(* Logix 5000 project; controller R5_CSS vendor 1 type 14 code 74 rev 19.11; software revision 19.01; part 7 of 20 *)
(* tags used below, declared in another part *)
   AC102A : ANALYTICAL;   // QUENCH WATER CONDUCTIVITY CONTROL
   AC102A_BLEED_MAKEUP_STATUS : DINT;   // 0=stopped 1=bleed water 2=makeup water 3=wait
   AC102A_BLEED_START_TON : TIMER;
   AC102A_BLEED_STOP_TON : TIMER;
   AC102A_BLEED_WAIT : BOOL;
   AC102A_BLEED_WAIT_TON : TIMER;
   AC102A_MAKEUP_STOP_TON : TIMER;
   AlarmMaster : DINT;
   AlarmsAckAll : BOOL;
   AlarmsDisabled : BOOL;
   F1_LC370 : LEVEL_CONTROL;
   FC141 : PUMP_CONTROL;
   FC215 : FLOW_CONTROL;   // OVERHEAD CONDENSER CHILLED WATER FLOW CONTROL
   FC365 : FLOW_CONTROL;   // COALESCER PROCESS IMPURITY FLOW CONTROL
   FC365_Alm : ALARM_ANALOG;
   FC365_AUTO_ONS1 : BOOL;
   FC365_AUTO_ONS2 : BOOL;
   FC365_BLEED_ALARM_DISABLE : BOOL;
   FC365_BLEED_FLOW_MIN_SP : DINT;
   FC365_BLEED_WAIT_MIN_SP : DINT;
   FC365_FLOW_TOO_LONG_ALM : BOOL;
   FC365_FLOW_TOO_LONG_RESETPB : BOOL;
   FC365_FLOW_TOO_LONG_TMR : TIMER;
   FC365_HMI_BLEED_START_ENABLE : BOOL;
   FC365_HMI_BLEED_START_ENABLE_TON : TIMER;
   FC365_HMI_BLEED_START_PB : BOOL;
   FC365_HMI_BLEED_STOP_PB : BOOL;
   FC365_LC370_FLOW_AUTO_SP : REAL;
   FC365_MANUAL_ONS1 : BOOL;
   FC365_MAX_TIME_MIN : DINT;
   FC365_Started : BOOL;
   FC365_TOTAl_GAL : REAL;
   FC365_TOTAl_RESET : BOOL;
   FC365_TOTAl_RESET_PB : BOOL;
   FC365_TOTALIZE : Totalize;
   FC365_TOTALIZE_EN : BOOL;
   FC365_TOTALIZE_EN_ONS1 : BOOL;
   FC365_TOTALIZE_LastFeedTimeMin : REAL;
   FC365_TOTALIZE_Min : REAL;
   FC365_TOTALIZE_TON : TIMER;
   FC365_UNABLE_TO_BLEED : BOOL;
   FC370 : FLOW_CONTROL;   // COALESCER MAKE UP WATER FLOW CONTROL
   FC403 : FLOW_CONTROL;   // COALESCER FLOW CONTROLLER FEEDS TCV108
   FC406 : FLOW_CONTROL;   // HX COOLING WATER FLOW CONTROL
   FCV141_MaxOpenSecSP : REAL;
   FCV141_MaxOpenTmr : TIMER;
   FireFlowAlarmFromUTL : BOOL;
   HS141 : ValveControl_TwoWay;
   InputMax_IF8 : REAL;
   InputMin_IF8 : REAL;
   LC303A : LEVEL_CONTROL;   // AQUEOUS PHASE OF PRIMARY SETTLER
   LC303B : LEVEL_CONTROL;   // INTERFACE LEVEL OF PRIMARY CONDENSER
   LC365_AUTO_SP_START : REAL;
   LC365_BLEED_AUTO_START : BOOL;
   LC365_BLEED_AUTO_START_TON : TIMER;
   LC365_LT : REAL;
   LC370 : LEVEL_CONTROL;   // WATER MAKE UP FOR PRIMARY SETTLER
   LC370_AUTO_SP_START : REAL;
   LCV370_Start : BOOL;
   PID_FCV365 : PID;
   PID_FCV365_TON : TIMER;
   PID_LC370_Enable : BOOL;
   SignalLossHigh_IF8 : DINT;
   SignalLossLow_IF8 : DINT;
   TC313A : TEMP_CONTROL;   // PRIMARY COALESCER SEPARATOR TEMPERATURE CONTROL
   TMR_FAULT : DINT;
   UTL_Comms : DINT[3];
(* MainProgram, continued *)

ROUTINE FC215_OverheadCondChillWaterFlow   (* ladder *)
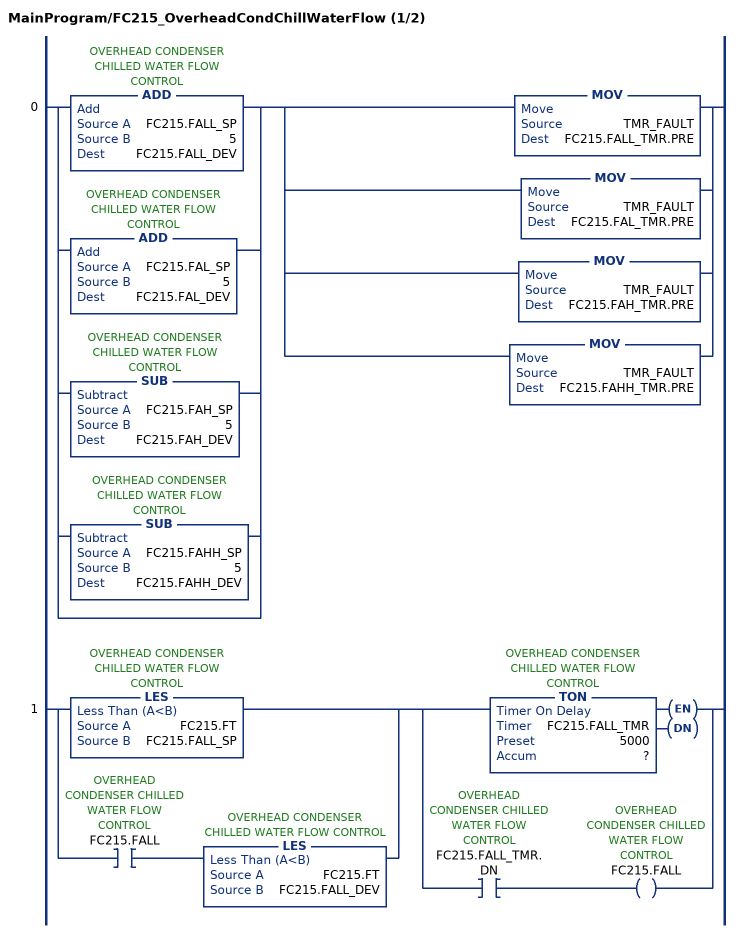
   0: [ADD(FC215.FALL_SP,5,FC215.FALL_DEV) ,ADD(FC215.FAL_SP,5,FC215.FAL_DEV) ,SUB(FC215.FAH_SP,5,FC215.FAH_DEV) ,SUB(FC215.FAHH_SP,5,FC215.FAHH_DEV) ,][MOV(TMR_FAULT,FC215.FALL_TMR.PRE) ,MOV(TMR_FAULT,FC215.FAL_TMR.PRE) ,MOV(TMR_FAULT,FC215.FAH_TMR.PRE) ,MOV(TMR_FAULT,FC215.FAHH_TMR.PRE) ];
   1: [LES(FC215.FT,FC215.FALL_SP) ,XIC(FC215.FALL) LES(FC215.FT,FC215.FALL_DEV) ][TON(FC215.FALL_TMR,?,?) ,XIC(FC215.FALL_TMR.DN) OTE(FC215.FALL) ];
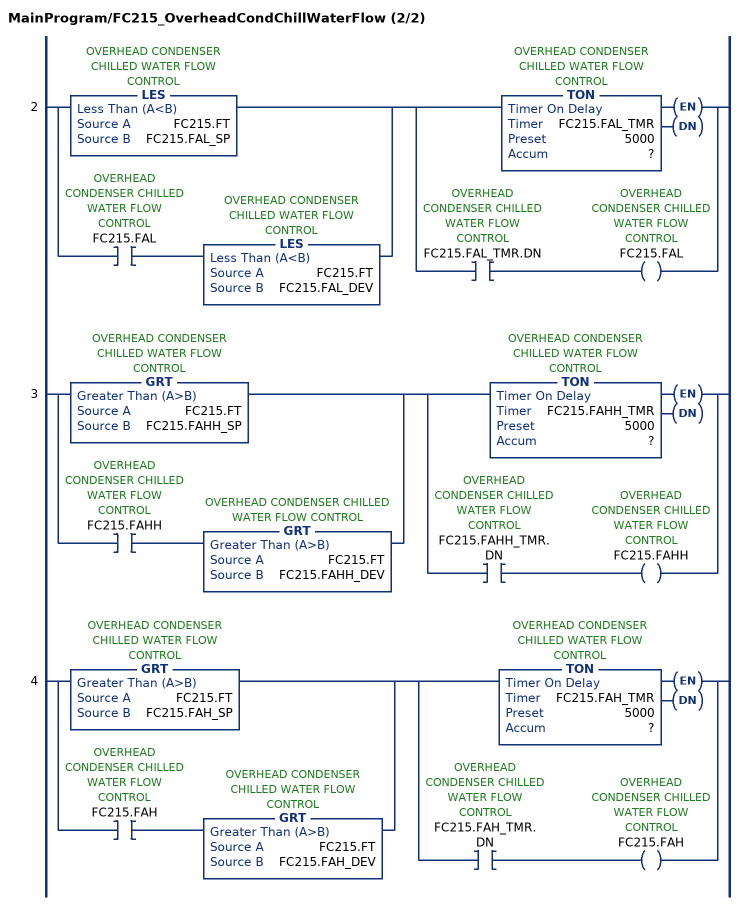
   2: [LES(FC215.FT,FC215.FAL_SP) ,XIC(FC215.FAL) LES(FC215.FT,FC215.FAL_DEV) ][TON(FC215.FAL_TMR,?,?) ,XIC(FC215.FAL_TMR.DN) OTE(FC215.FAL) ];
   3: [GRT(FC215.FT,FC215.FAHH_SP) ,XIC(FC215.FAHH) GRT(FC215.FT,FC215.FAHH_DEV) ][TON(FC215.FAHH_TMR,?,?) ,XIC(FC215.FAHH_TMR.DN) OTE(FC215.FAHH) ];
   4: [GRT(FC215.FT,FC215.FAH_SP) ,XIC(FC215.FAH) GRT(FC215.FT,FC215.FAH_DEV) ][TON(FC215.FAH_TMR,?,?) ,XIC(FC215.FAH_TMR.DN) OTE(FC215.FAH) ];
END_ROUTINE

ROUTINE FC370_WaterMakeupFlow   (* ladder *)
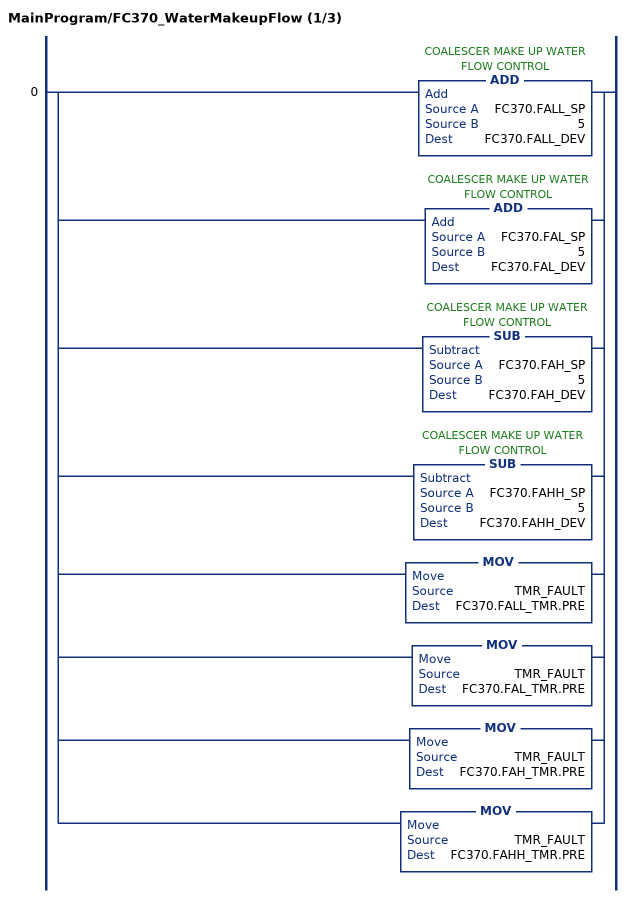
   0: [ADD(FC370.FALL_SP,5,FC370.FALL_DEV) ,ADD(FC370.FAL_SP,5,FC370.FAL_DEV) ,SUB(FC370.FAH_SP,5,FC370.FAH_DEV) ,SUB(FC370.FAHH_SP,5,FC370.FAHH_DEV) ,MOV(TMR_FAULT,FC370.FALL_TMR.PRE) ,MOV(TMR_FAULT,FC370.FAL_TMR.PRE) ,MOV(TMR_FAULT,FC370.FAH_TMR.PRE) ,MOV(TMR_FAULT,FC370.FAHH_TMR.PRE) ];
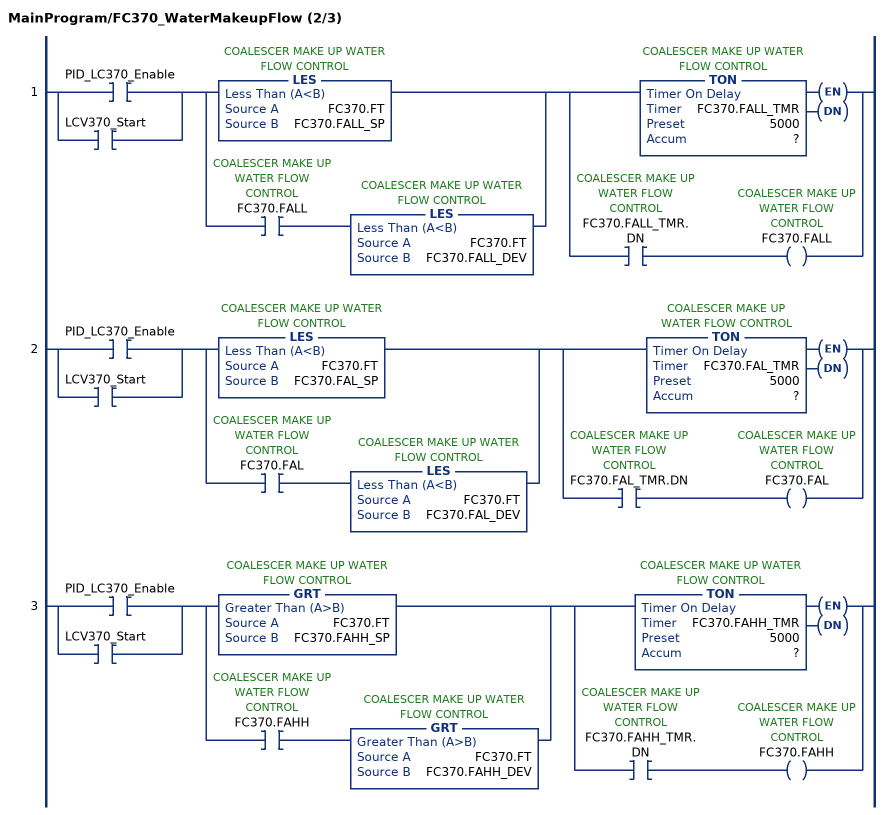
   1: [XIC(PID_LC370_Enable) ,XIC(LCV370_Start) ][LES(FC370.FT,FC370.FALL_SP) ,XIC(FC370.FALL) LES(FC370.FT,FC370.FALL_DEV) ][TON(FC370.FALL_TMR,?,?) ,XIC(FC370.FALL_TMR.DN) OTE(FC370.FALL) ];
   2: [XIC(PID_LC370_Enable) ,XIC(LCV370_Start) ][LES(FC370.FT,FC370.FAL_SP) ,XIC(FC370.FAL) LES(FC370.FT,FC370.FAL_DEV) ][TON(FC370.FAL_TMR,?,?) ,XIC(FC370.FAL_TMR.DN) OTE(FC370.FAL) ];
   3: [XIC(PID_LC370_Enable) ,XIC(LCV370_Start) ][GRT(FC370.FT,FC370.FAHH_SP) ,XIC(FC370.FAHH) GRT(FC370.FT,FC370.FAHH_DEV) ][TON(FC370.FAHH_TMR,?,?) ,XIC(FC370.FAHH_TMR.DN) OTE(FC370.FAHH) ];
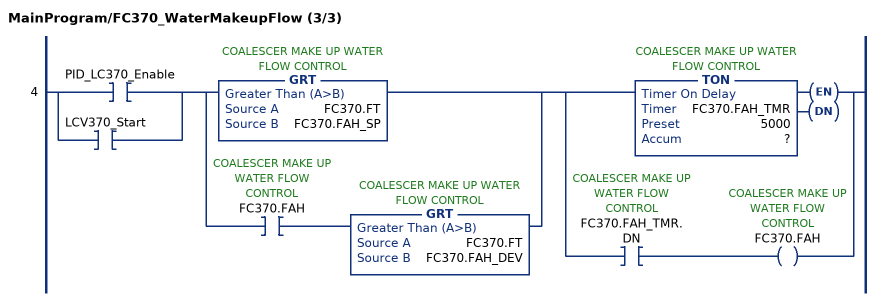
   4: [XIC(PID_LC370_Enable) ,XIC(LCV370_Start) ][GRT(FC370.FT,FC370.FAH_SP) ,XIC(FC370.FAH) GRT(FC370.FT,FC370.FAH_DEV) ][TON(FC370.FAH_TMR,?,?) ,XIC(FC370.FAH_TMR.DN) OTE(FC370.FAH) ];
END_ROUTINE

ROUTINE FC403_QuenchWaterTotalFlow   (* ladder *)
// COALESCER FLOW CONTROL
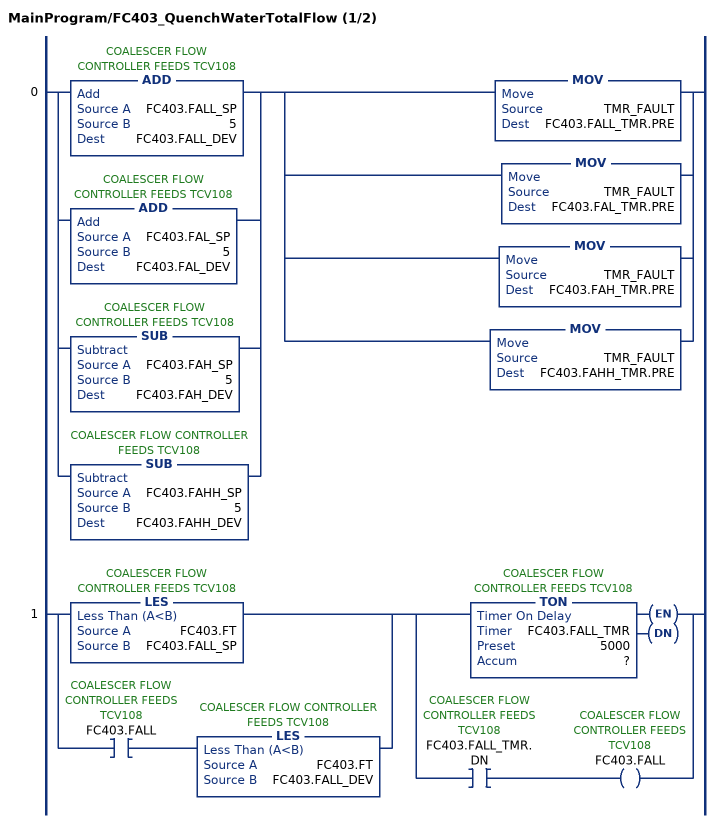
   0: [ADD(FC403.FALL_SP,5,FC403.FALL_DEV) ,ADD(FC403.FAL_SP,5,FC403.FAL_DEV) ,SUB(FC403.FAH_SP,5,FC403.FAH_DEV) ,SUB(FC403.FAHH_SP,5,FC403.FAHH_DEV) ][MOV(TMR_FAULT,FC403.FALL_TMR.PRE) ,MOV(TMR_FAULT,FC403.FAL_TMR.PRE) ,MOV(TMR_FAULT,FC403.FAH_TMR.PRE) ,MOV(TMR_FAULT,FC403.FAHH_TMR.PRE) ];
   1: [LES(FC403.FT,FC403.FALL_SP) ,XIC(FC403.FALL) LES(FC403.FT,FC403.FALL_DEV) ][TON(FC403.FALL_TMR,?,?) ,XIC(FC403.FALL_TMR.DN) OTE(FC403.FALL) ];
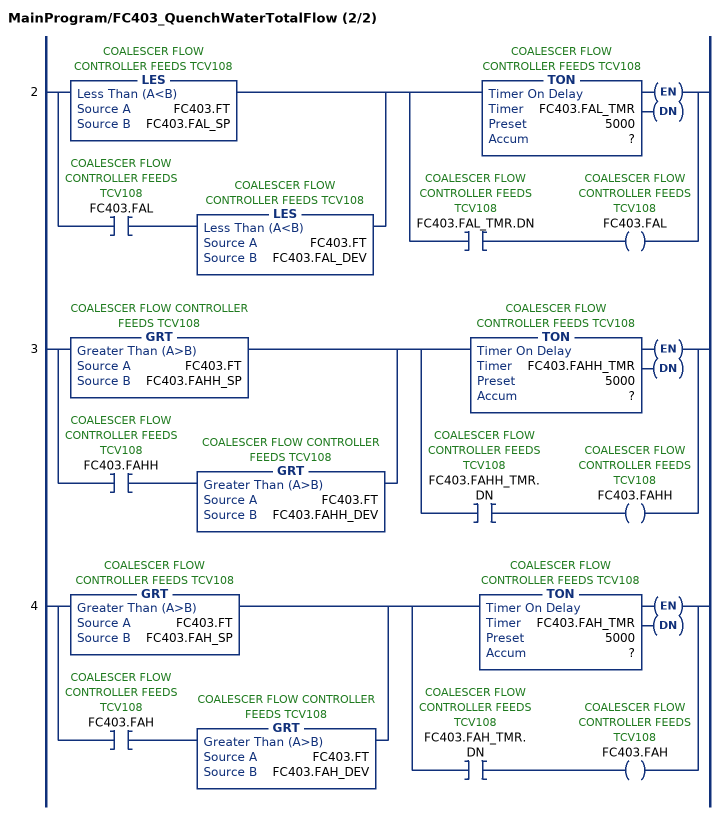
   2: [LES(FC403.FT,FC403.FAL_SP) ,XIC(FC403.FAL) LES(FC403.FT,FC403.FAL_DEV) ][TON(FC403.FAL_TMR,?,?) ,XIC(FC403.FAL_TMR.DN) OTE(FC403.FAL) ];
   3: [GRT(FC403.FT,FC403.FAHH_SP) ,XIC(FC403.FAHH) GRT(FC403.FT,FC403.FAHH_DEV) ][TON(FC403.FAHH_TMR,?,?) ,XIC(FC403.FAHH_TMR.DN) OTE(FC403.FAHH) ];
   4: [GRT(FC403.FT,FC403.FAH_SP) ,XIC(FC403.FAH) GRT(FC403.FT,FC403.FAH_DEV) ][TON(FC403.FAH_TMR,?,?) ,XIC(FC403.FAH_TMR.DN) OTE(FC403.FAH) ];
END_ROUTINE

ROUTINE FC406_CoolingWaterFlow   (* ladder *)
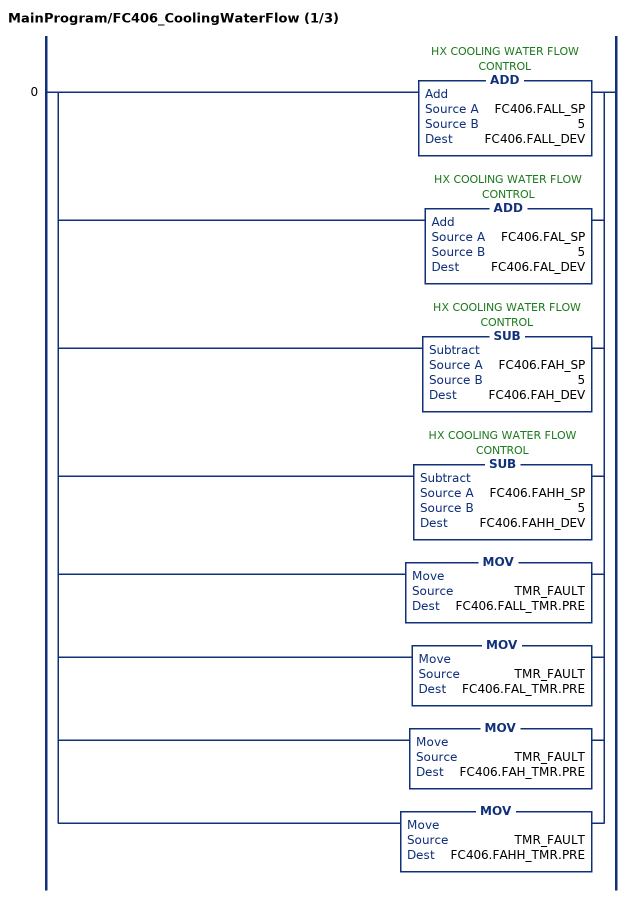
   0: [ADD(FC406.FALL_SP,5,FC406.FALL_DEV) ,ADD(FC406.FAL_SP,5,FC406.FAL_DEV) ,SUB(FC406.FAH_SP,5,FC406.FAH_DEV) ,SUB(FC406.FAHH_SP,5,FC406.FAHH_DEV) ,MOV(TMR_FAULT,FC406.FALL_TMR.PRE) ,MOV(TMR_FAULT,FC406.FAL_TMR.PRE) ,MOV(TMR_FAULT,FC406.FAH_TMR.PRE) ,MOV(TMR_FAULT,FC406.FAHH_TMR.PRE) ];
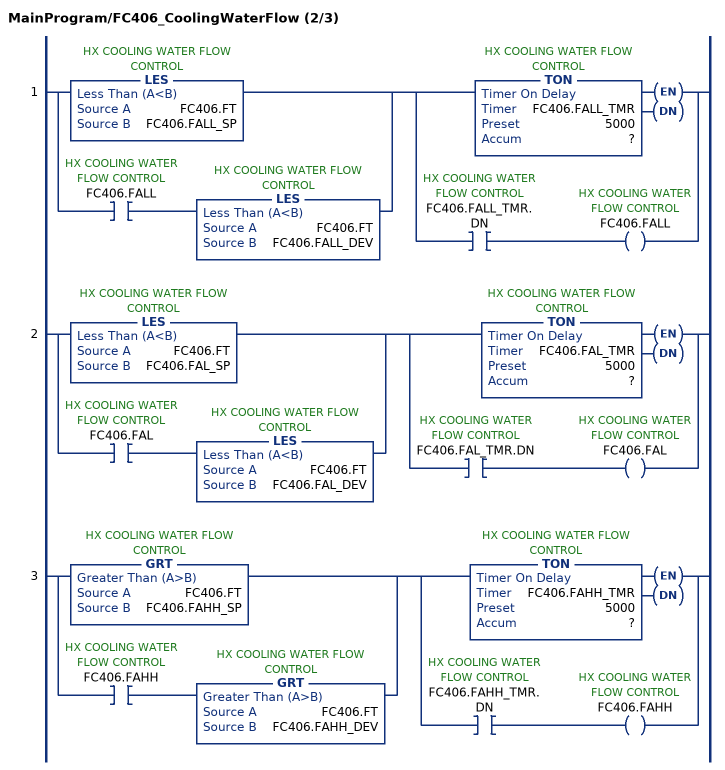
   1: [LES(FC406.FT,FC406.FALL_SP) ,XIC(FC406.FALL) LES(FC406.FT,FC406.FALL_DEV) ][TON(FC406.FALL_TMR,?,?) ,XIC(FC406.FALL_TMR.DN) OTE(FC406.FALL) ];
   2: [LES(FC406.FT,FC406.FAL_SP) ,XIC(FC406.FAL) LES(FC406.FT,FC406.FAL_DEV) ][TON(FC406.FAL_TMR,?,?) ,XIC(FC406.FAL_TMR.DN) OTE(FC406.FAL) ];
   3: [GRT(FC406.FT,FC406.FAHH_SP) ,XIC(FC406.FAHH) GRT(FC406.FT,FC406.FAHH_DEV) ][TON(FC406.FAHH_TMR,?,?) ,XIC(FC406.FAHH_TMR.DN) OTE(FC406.FAHH) ];
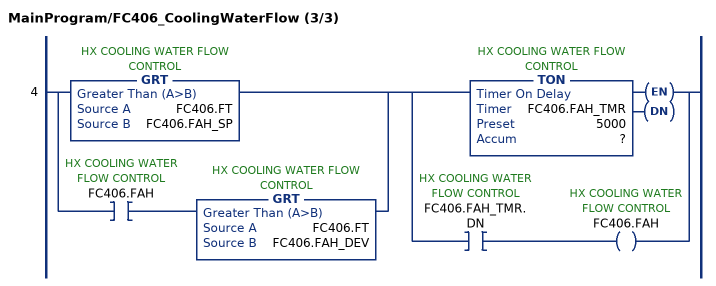
   4: [GRT(FC406.FT,FC406.FAH_SP) ,XIC(FC406.FAH) GRT(FC406.FT,FC406.FAH_DEV) ][TON(FC406.FAH_TMR,?,?) ,XIC(FC406.FAH_TMR.DN) OTE(FC406.FAH) ];
END_ROUTINE

ROUTINE FCV141_QuenchTowerEmegencyValve   (* ladder *)
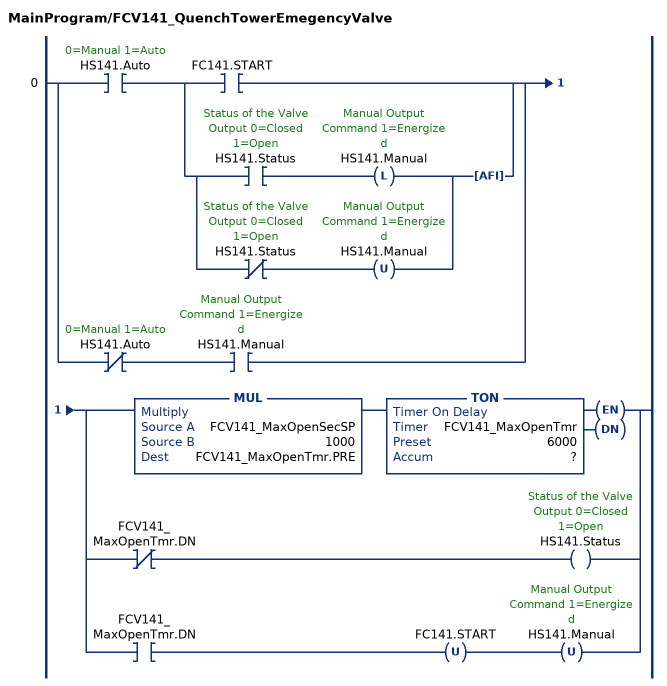
   0: [XIC(HS141.Auto) [XIC(FC141.START) ,[XIC(HS141.Status) OTL(HS141.Manual) ,XIO(HS141.Status) OTU(HS141.Manual) ] AFI() ] ,XIO(HS141.Auto) XIC(HS141.Manual) ][MUL(FCV141_MaxOpenSecSP,1000,FCV141_MaxOpenTmr.PRE) TON(FCV141_MaxOpenTmr,?,?) ,XIO(FCV141_MaxOpenTmr.DN) OTE(HS141.Status) ,XIC(FCV141_MaxOpenTmr.DN) OTU(FC141.START) OTU(HS141.Manual) ];
END_ROUTINE

ROUTINE FCV365_WaterBleedLevel_PID   (* ladder *)
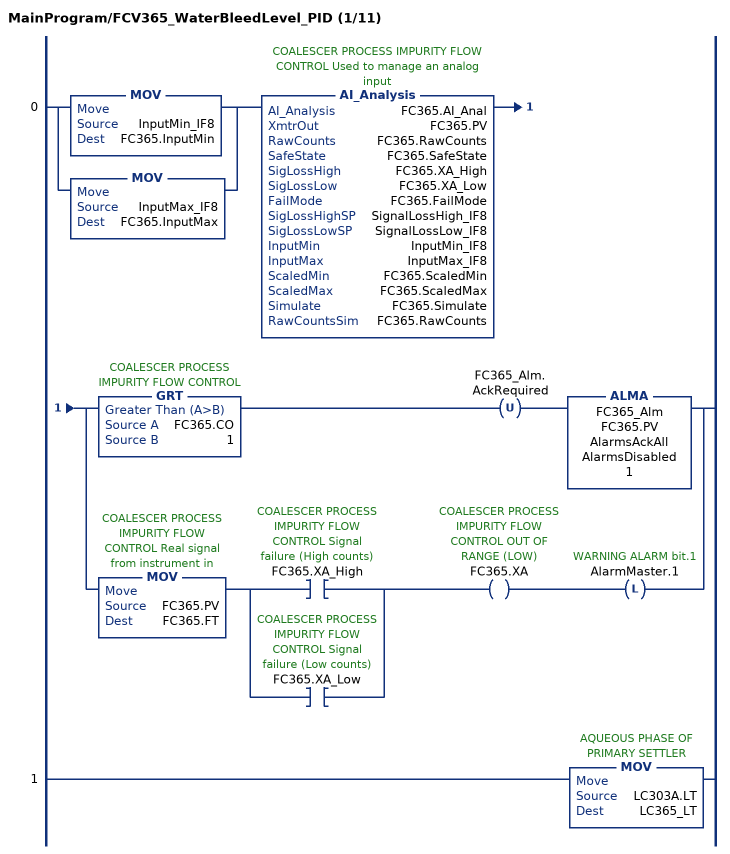
   0: [MOV(InputMin_IF8,FC365.InputMin) ,MOV(InputMax_IF8,FC365.InputMax) ]AI_Analysis(FC365.AI_Anal,FC365.PV,FC365.RawCounts,FC365.SafeState,FC365.XA_High,FC365.XA_Low,FC365.FailMode,SignalLossHigh_IF8,SignalLossLow_IF8,InputMin_IF8,InputMax_IF8,FC365.ScaledMin,FC365.ScaledMax,FC365.Simulate,FC365.RawCounts)[GRT(FC365.CO,1) OTU(FC365_Alm.AckRequired) ALMA(FC365_Alm,FC365.PV,AlarmsAckAll,AlarmsDisabled,1) ,MOV(FC365.PV,FC365.FT) [XIC(FC365.XA_High) ,XIC(FC365.XA_Low) ] OTE(FC365.XA) OTL(AlarmMaster.1) ];
   1: MOV(LC303A.LT,LC365_LT);
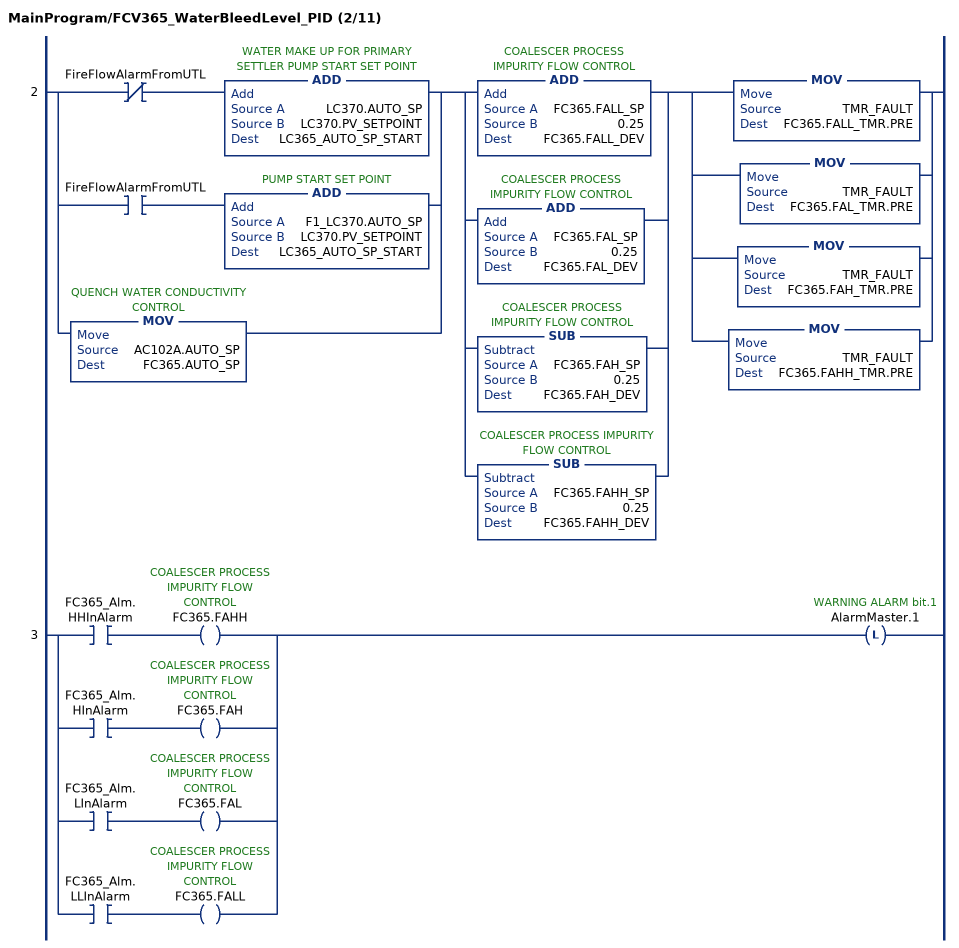
   2: [XIO(FireFlowAlarmFromUTL) ADD(LC370.AUTO_SP,LC370.PV_SETPOINT,LC365_AUTO_SP_START) ,XIC(FireFlowAlarmFromUTL) ADD(F1_LC370.AUTO_SP,LC370.PV_SETPOINT,LC365_AUTO_SP_START) ,MOV(AC102A.AUTO_SP,FC365.AUTO_SP) ][ADD(FC365.FALL_SP,0.25,FC365.FALL_DEV) ,ADD(FC365.FAL_SP,0.25,FC365.FAL_DEV) ,SUB(FC365.FAH_SP,0.25,FC365.FAH_DEV) ,SUB(FC365.FAHH_SP,0.25,FC365.FAHH_DEV) ][MOV(TMR_FAULT,FC365.FALL_TMR.PRE) ,MOV(TMR_FAULT,FC365.FAL_TMR.PRE) ,MOV(TMR_FAULT,FC365.FAH_TMR.PRE) ,MOV(TMR_FAULT,FC365.FAHH_TMR.PRE) ];
   3: [XIC(FC365_Alm.HHInAlarm) OTE(FC365.FAHH) ,XIC(FC365_Alm.HInAlarm) OTE(FC365.FAH) ,XIC(FC365_Alm.LInAlarm) OTE(FC365.FAL) ,XIC(FC365_Alm.LLInAlarm) OTE(FC365.FALL) ]OTL(AlarmMaster.1);
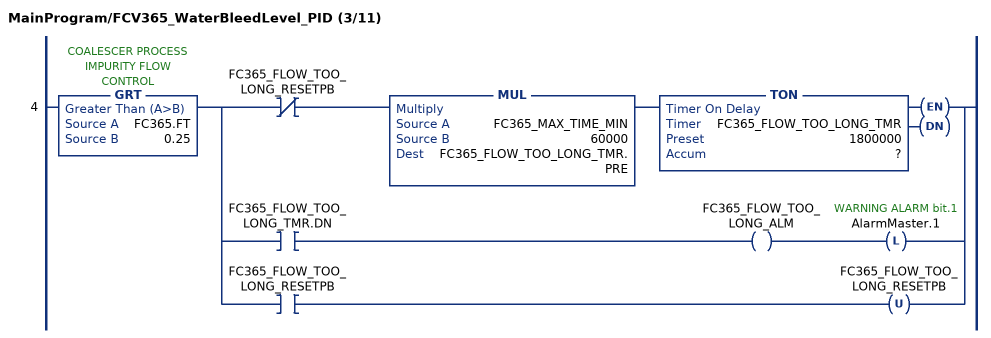
   4: GRT(FC365.FT,0.25)[XIO(FC365_FLOW_TOO_LONG_RESETPB) MUL(FC365_MAX_TIME_MIN,60000,FC365_FLOW_TOO_LONG_TMR.PRE) TON(FC365_FLOW_TOO_LONG_TMR,?,?) ,XIC(FC365_FLOW_TOO_LONG_TMR.DN) OTE(FC365_FLOW_TOO_LONG_ALM) OTL(AlarmMaster.1) ,XIC(FC365_FLOW_TOO_LONG_RESETPB) OTU(FC365_FLOW_TOO_LONG_RESETPB) ];
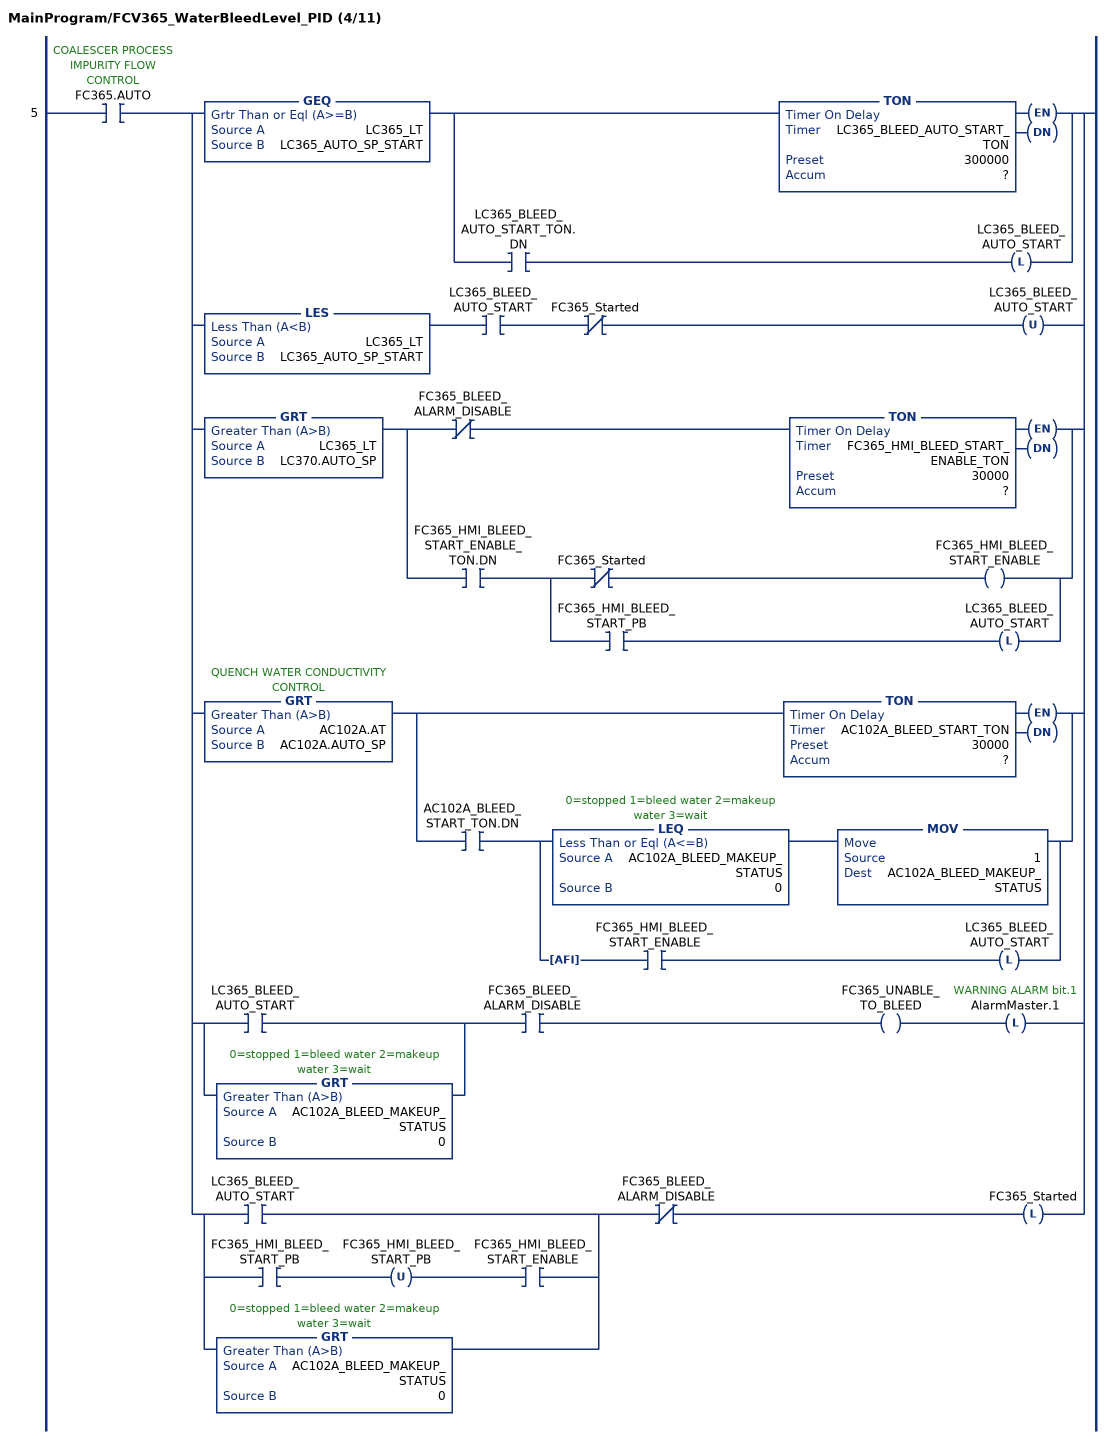
   5: XIC(FC365.AUTO)[GEQ(LC365_LT,LC365_AUTO_SP_START) [TON(LC365_BLEED_AUTO_START_TON,?,?) ,XIC(LC365_BLEED_AUTO_START_TON.DN) OTL(LC365_BLEED_AUTO_START) ] ,LES(LC365_LT,LC365_AUTO_SP_START) XIC(LC365_BLEED_AUTO_START) XIO(FC365_Started) OTU(LC365_BLEED_AUTO_START) ,GRT(LC365_LT,LC370.AUTO_SP) [XIO(FC365_BLEED_ALARM_DISABLE) TON(FC365_HMI_BLEED_START_ENABLE_TON,?,?) ,XIC(FC365_HMI_BLEED_START_ENABLE_TON.DN) [XIO(FC365_Started) OTE(FC365_HMI_BLEED_START_ENABLE) ,XIC(FC365_HMI_BLEED_START_PB) OTL(LC365_BLEED_AUTO_START) ] ] ,GRT(AC102A.AT,AC102A.AUTO_SP) [TON(AC102A_BLEED_START_TON,?,?) ,XIC(AC102A_BLEED_START_TON.DN) [LEQ(AC102A_BLEED_MAKEUP_STATUS,0) MOV(1,AC102A_BLEED_MAKEUP_STATUS) ,AFI() XIC(FC365_HMI_BLEED_START_ENABLE) OTL(LC365_BLEED_AUTO_START) ] ] ,[XIC(LC365_BLEED_AUTO_START) ,GRT(AC102A_BLEED_MAKEUP_STATUS,0) ] XIC(FC365_BLEED_ALARM_DISABLE) OTE(FC365_UNABLE_TO_BLEED) OTL(AlarmMaster.1) ,[XIC(LC365_BLEED_AUTO_START) ,XIC(FC365_HMI_BLEED_START_PB) OTU(FC365_HMI_BLEED_START_PB) XIC(FC365_HMI_BLEED_START_ENABLE) ,GRT(AC102A_BLEED_MAKEUP_STATUS,0) ] XIO(FC365_BLEED_ALARM_DISABLE) OTL(FC365_Started) ];
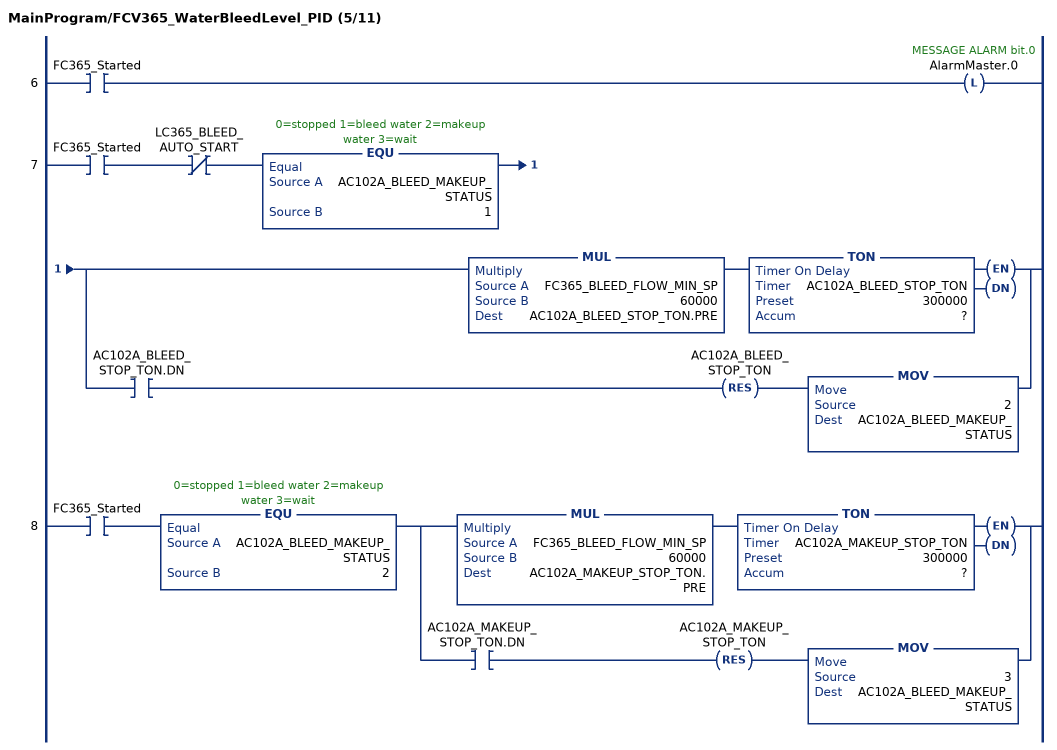
   6: XIC(FC365_Started)OTL(AlarmMaster.0);
   7: XIC(FC365_Started)XIO(LC365_BLEED_AUTO_START)EQU(AC102A_BLEED_MAKEUP_STATUS,1)[MUL(FC365_BLEED_FLOW_MIN_SP,60000,AC102A_BLEED_STOP_TON.PRE) TON(AC102A_BLEED_STOP_TON,?,?) ,XIC(AC102A_BLEED_STOP_TON.DN) RES(AC102A_BLEED_STOP_TON) MOV(2,AC102A_BLEED_MAKEUP_STATUS) ];
   8: XIC(FC365_Started)EQU(AC102A_BLEED_MAKEUP_STATUS,2)[MUL(FC365_BLEED_FLOW_MIN_SP,60000,AC102A_MAKEUP_STOP_TON.PRE) TON(AC102A_MAKEUP_STOP_TON,?,?) ,XIC(AC102A_MAKEUP_STOP_TON.DN) RES(AC102A_MAKEUP_STOP_TON) MOV(3,AC102A_BLEED_MAKEUP_STATUS) ];
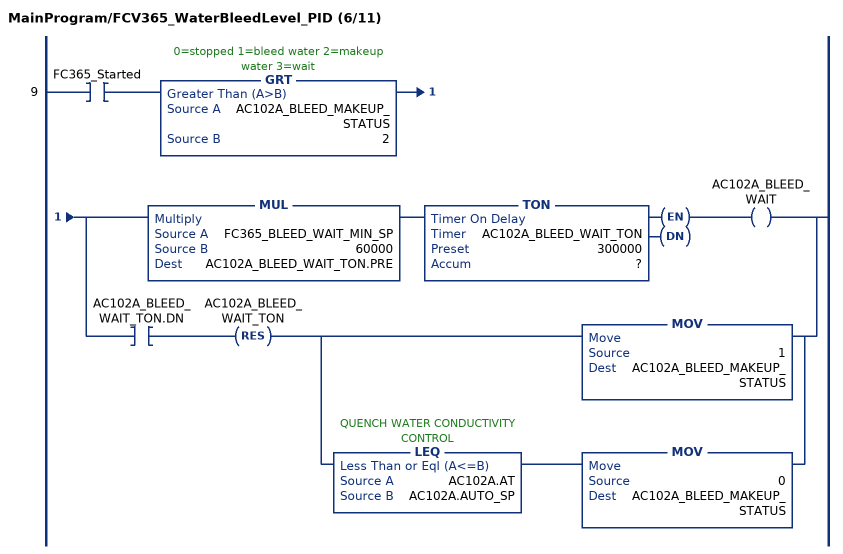
   9: XIC(FC365_Started)GRT(AC102A_BLEED_MAKEUP_STATUS,2)[MUL(FC365_BLEED_WAIT_MIN_SP,60000,AC102A_BLEED_WAIT_TON.PRE) TON(AC102A_BLEED_WAIT_TON,?,?) OTE(AC102A_BLEED_WAIT) ,XIC(AC102A_BLEED_WAIT_TON.DN) RES(AC102A_BLEED_WAIT_TON) [MOV(1,AC102A_BLEED_MAKEUP_STATUS) ,LEQ(AC102A.AT,AC102A.AUTO_SP) MOV(0,AC102A_BLEED_MAKEUP_STATUS) ] ];
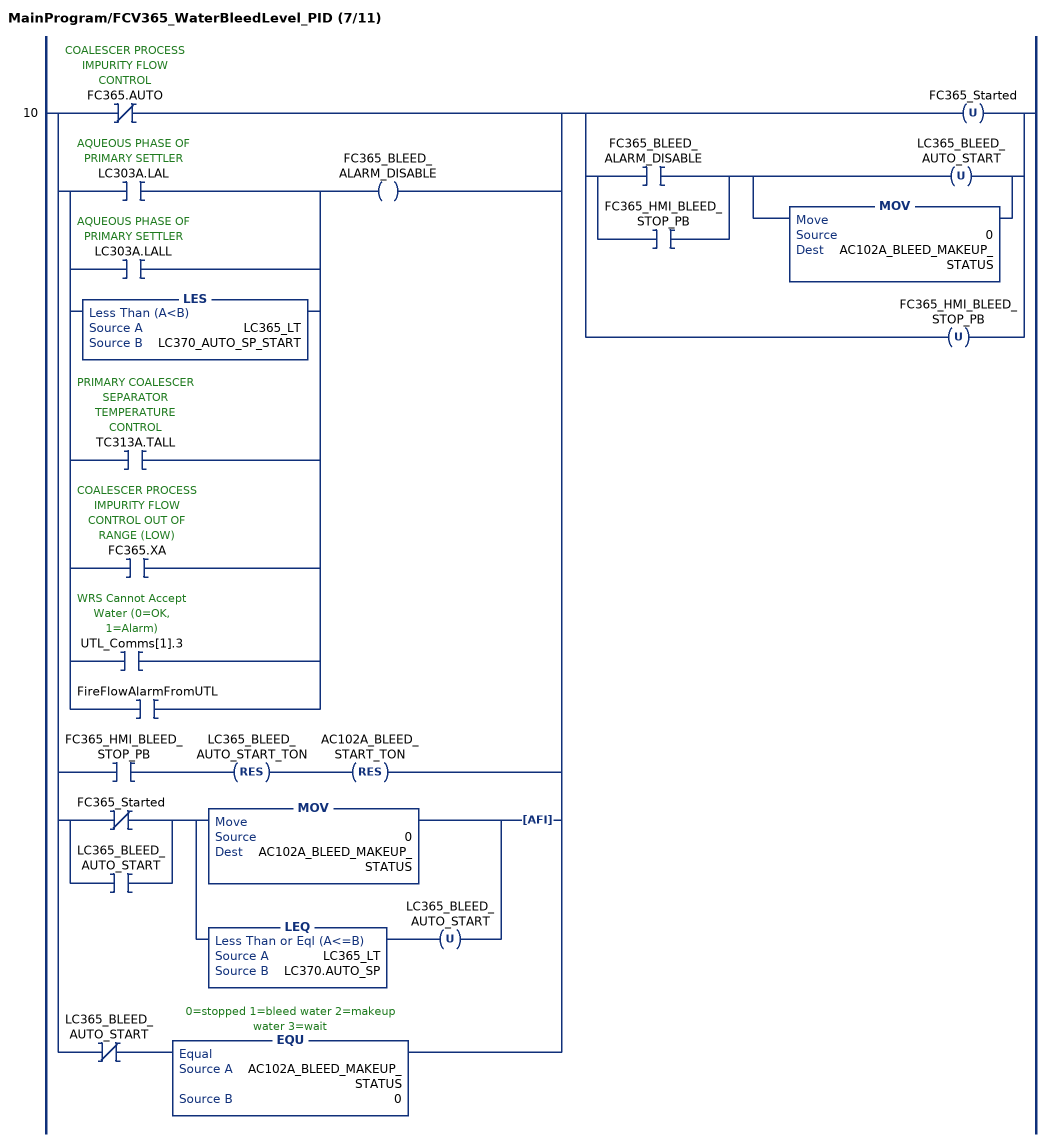
   10: [XIO(FC365.AUTO) ,[XIC(LC303A.LAL) ,XIC(LC303A.LALL) ,LES(LC365_LT,LC370_AUTO_SP_START) ,XIC(TC313A.TALL) ,XIC(FC365.XA) ,XIC(UTL_Comms[1].3) ,XIC(FireFlowAlarmFromUTL) ] OTE(FC365_BLEED_ALARM_DISABLE) ,XIC(FC365_HMI_BLEED_STOP_PB) RES(LC365_BLEED_AUTO_START_TON) RES(AC102A_BLEED_START_TON) ,[XIO(FC365_Started) ,XIC(LC365_BLEED_AUTO_START) ] [MOV(0,AC102A_BLEED_MAKEUP_STATUS) ,LEQ(LC365_LT,LC370.AUTO_SP) OTU(LC365_BLEED_AUTO_START) ] AFI() ,XIO(LC365_BLEED_AUTO_START) EQU(AC102A_BLEED_MAKEUP_STATUS,0) ][OTU(FC365_Started) ,[XIC(FC365_BLEED_ALARM_DISABLE) ,XIC(FC365_HMI_BLEED_STOP_PB) ] [OTU(LC365_BLEED_AUTO_START) ,MOV(0,AC102A_BLEED_MAKEUP_STATUS) ] ,OTU(FC365_HMI_BLEED_STOP_PB) ];
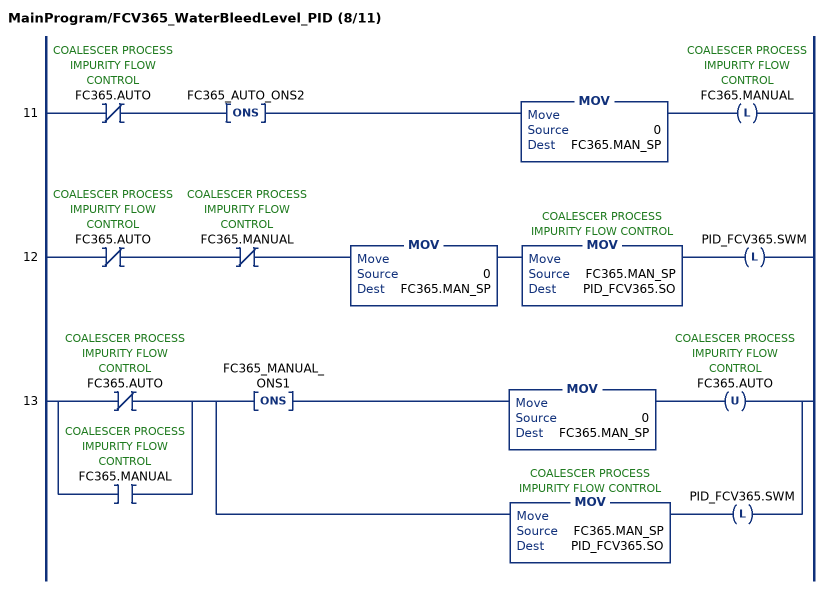
   11: XIO(FC365.AUTO)ONS(FC365_AUTO_ONS2)MOV(0,FC365.MAN_SP)OTL(FC365.MANUAL);
   12: XIO(FC365.AUTO)XIO(FC365.MANUAL)MOV(0,FC365.MAN_SP)MOV(FC365.MAN_SP,PID_FCV365.SO)OTL(PID_FCV365.SWM);
   13: [XIO(FC365.AUTO) ,XIC(FC365.MANUAL) ][ONS(FC365_MANUAL_ONS1) MOV(0,FC365.MAN_SP) OTU(FC365.AUTO) ,MOV(FC365.MAN_SP,PID_FCV365.SO) OTL(PID_FCV365.SWM) ];
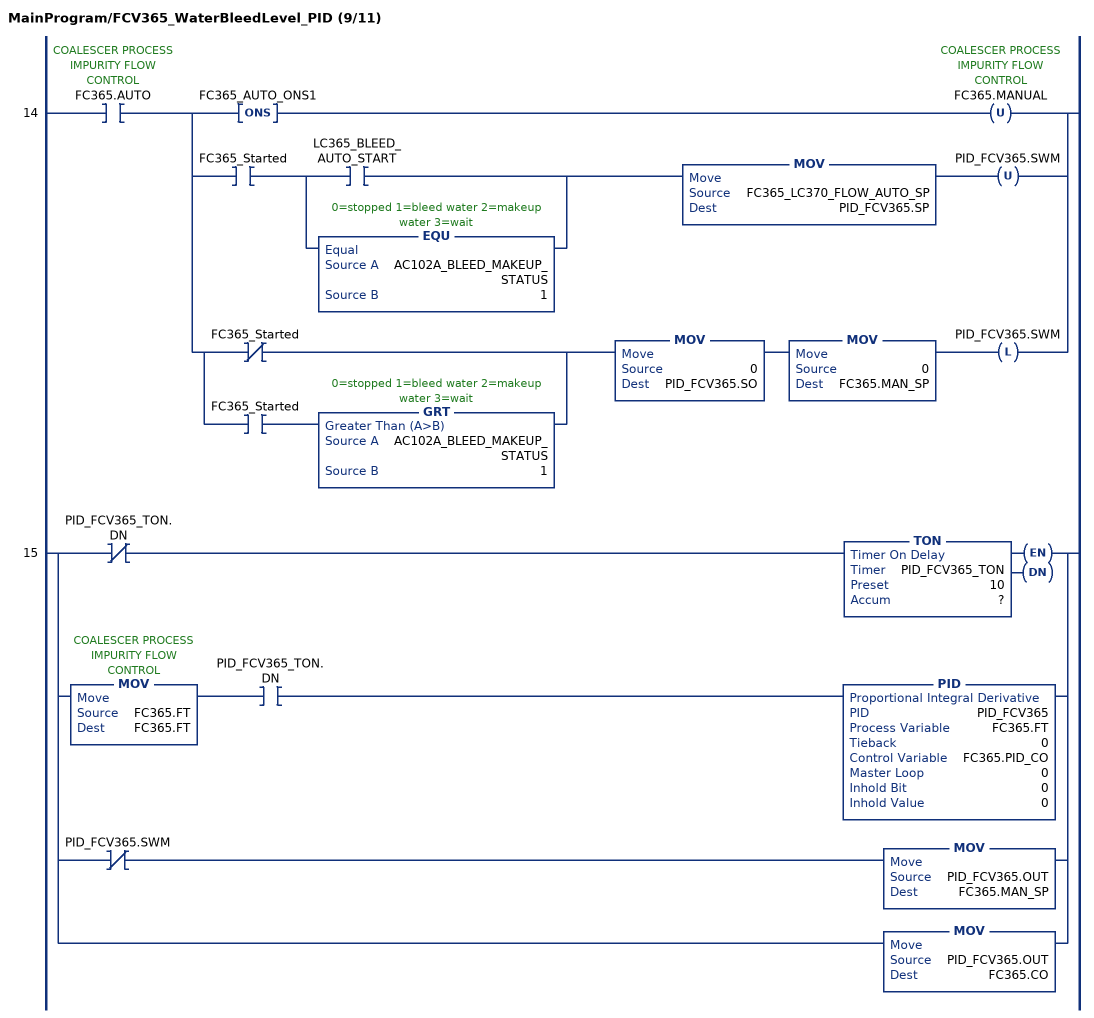
   14: XIC(FC365.AUTO)[ONS(FC365_AUTO_ONS1) OTU(FC365.MANUAL) ,XIC(FC365_Started) [XIC(LC365_BLEED_AUTO_START) ,EQU(AC102A_BLEED_MAKEUP_STATUS,1) ] MOV(FC365_LC370_FLOW_AUTO_SP,PID_FCV365.SP) OTU(PID_FCV365.SWM) ,[XIO(FC365_Started) ,XIC(FC365_Started) GRT(AC102A_BLEED_MAKEUP_STATUS,1) ] MOV(0,PID_FCV365.SO) MOV(0,FC365.MAN_SP) OTL(PID_FCV365.SWM) ];
   15: [XIO(PID_FCV365_TON.DN) TON(PID_FCV365_TON,?,?) ,MOV(FC365.FT,FC365.FT) XIC(PID_FCV365_TON.DN) PID(PID_FCV365,FC365.FT,0,FC365.PID_CO,0,0,0) ,XIO(PID_FCV365.SWM) MOV(PID_FCV365.OUT,FC365.MAN_SP) ,MOV(PID_FCV365.OUT,FC365.CO) ];
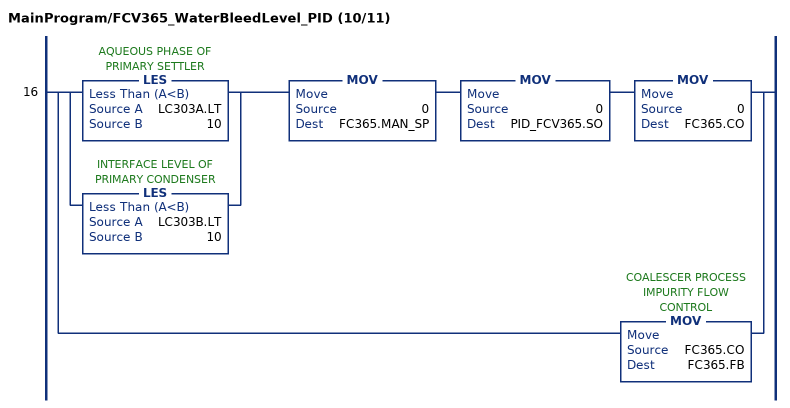
   16: [[LES(LC303A.LT,10) ,LES(LC303B.LT,10) ] MOV(0,FC365.MAN_SP) MOV(0,PID_FCV365.SO) MOV(0,FC365.CO) ,MOV(FC365.CO,FC365.FB) ];
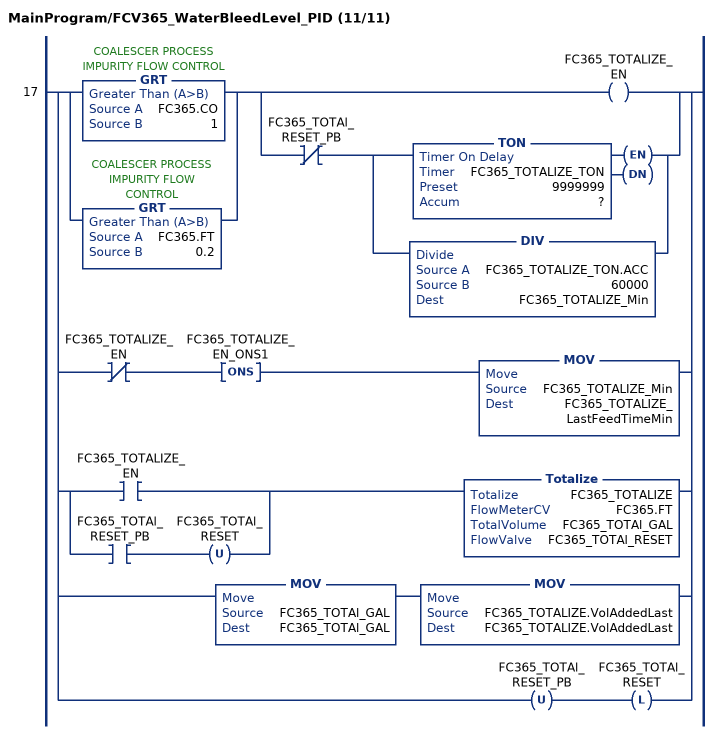
   17: [[GRT(FC365.CO,1) ,GRT(FC365.FT,0.2) ] [OTE(FC365_TOTALIZE_EN) ,XIO(FC365_TOTAl_RESET_PB) [TON(FC365_TOTALIZE_TON,?,?) ,DIV(FC365_TOTALIZE_TON.ACC,60000,FC365_TOTALIZE_Min) ] ] ,XIO(FC365_TOTALIZE_EN) ONS(FC365_TOTALIZE_EN_ONS1) MOV(FC365_TOTALIZE_Min,FC365_TOTALIZE_LastFeedTimeMin) ,[XIC(FC365_TOTALIZE_EN) ,XIC(FC365_TOTAl_RESET_PB) OTU(FC365_TOTAl_RESET) ] Totalize(FC365_TOTALIZE,FC365.FT,FC365_TOTAl_GAL,FC365_TOTAl_RESET) ,MOV(FC365_TOTAl_GAL,FC365_TOTAl_GAL) MOV(FC365_TOTALIZE.VolAddedLast,FC365_TOTALIZE.VolAddedLast) ,OTU(FC365_TOTAl_RESET_PB) OTL(FC365_TOTAl_RESET) ];
END_ROUTINE
